FUNCTION_BLOCK GF_Pumpen EXTENDS FB_Basisfunktionalitaeten
VAR_INPUT
	// Instanzieren von Sensoren mit Interfaces
	
	// Instanzieren von Aktoren mit Interfaces
	
	
END_VAR
VAR_OUTPUT
	
END_VAR
VAR
	
END_VAR

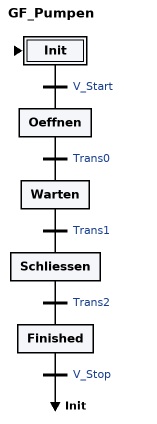
INITIAL_STEP Init:
END_STEP
TRANSITION FROM Init TO Oeffnen
    := V_Start;
END_TRANSITION
STEP Oeffnen:
END_STEP
TRANSITION FROM Oeffnen TO Warten
    := Trans0;
END_TRANSITION
STEP Warten:
END_STEP
TRANSITION FROM Warten TO Schliessen
    := Trans1;
END_TRANSITION
STEP Schliessen:
END_STEP
TRANSITION FROM Schliessen TO Finished
    := Trans2;
END_TRANSITION
STEP Finished:
END_STEP
TRANSITION FROM Finished TO Init
    := V_Stop;
END_TRANSITION

END_FUNCTION_BLOCK

(* stored: Version 1.1.0.1, ProductVersion 3.1.4024.12
   POU GF_Pumpen: Id {298b1c00-eb4e-4c76-a60a-3efaa29ca07f}, SpecialFunc None *)
